FUNCTION Convert_LWORD_TO_DINT : Hresult
VAR_INPUT
	in : LWORD;
	out : REFERENCE TO DINT;
END_VAR
VAR
	converted : DINT;
END_VAR

converted := LWORD_TO_DINT(in);

IF (DINT_TO_LWORD(converted) <> in) THEN
	Convert_LWORD_TO_DINT := INCOMPATIBLE;
	RETURN;
END_IF

out := converted;

END_FUNCTION

(* stored: Version 1.1.0.1, ProductVersion 3.1.4024.12
   POU Convert_LWORD_TO_DINT: Id {97acb6e4-976a-47c8-85db-597d9328d6fa}, SpecialFunc None *)
